(* PLC project CM, Beckhoff Automation GmbH TwinCAT PLC Control 3.5.13.21 *)
(* stored: creationDateTime 2024-07-22T16:12:49.8021823, modificationDateTime 2024-07-22T16:12:49.8062692 *)

TYPE E_AnalysisIDs :
(
	(* analysis chain *)
	eID_Source := 1,
	
	// Magnetude Spectrum
	eID_MagSpectrum,	
	eID_MagSpec_Sink, 
	
	// RMS intergrate
	eID_RMS,	
	eID_RMS_Sink,
	
	// Envelope Spectrum
	eID_EnvSpectrum,	
	eID_EnvSpec_Sink,
	
	// Envelope 
	eID_Env,	
	eID_Env_Sink	
	
) UDINT;
END_TYPE

TYPE ST_HRErrHist :
STRUCT
{attribute 'displaymode':='hex'}
	hrErrCode	: HRESULT;
	sErrSource	: STRING(63);
	nErrCount	: UDINT;
END_STRUCT
END_TYPE

FUNCTION_BLOCK FB_HRErrHist
(* v1.10
build up an error history consisting of two arrays and one index.
The index shows the actual array position. The last error id and the count for this id are saved in the arrays.
If an error id is the same as the previous input error the counter is increased. Otherwise the index is increased.
*)
VAR_INPUT
	bEdgeDetect	: BOOL;	(* FALSE: every input(bErr) is processed; TRUE: only rising edge of input is processed *)
END_VAR
VAR_OUTPUT
	nErrSum		: UINT;
	nErrIdx		: UINT; // error list index of last occured error (max. cHistLen)
	aErrList	: ARRAY[1..cHistLen] OF ST_HRErrHist;
END_VAR

VAR
	bNewErr		: BOOL;
	fbErrTrig	: R_TRIG;
END_VAR
VAR CONSTANT
	cHistLen	: UINT := 100;
END_VAR

                  
                

METHOD AddError
VAR_INPUT
	bErr		: BOOL;
	hrErrCode	: HRESULT;
	sErrSource	: STRING(63);
END_VAR
                        fbErrTrig(CLK:=bErr);
IF bEdgeDetect THEN
	bNewErr := fbErrTrig.Q;
ELSE
	bNewErr := bErr;
END_IF

IF bNewErr THEN
	nErrSum := nErrSum + 1;
	IF nErrIdx < cHistLen THEN
		IF nErrIdx = 0 THEN
			nErrIdx	:= nErrIdx + 1;
		ELSIF aErrList[nErrIdx].hrErrCode <> hrErrCode OR aErrList[nErrIdx].sErrSource <> sErrSource THEN
			nErrIdx	:= nErrIdx + 1;
		END_IF
		aErrList[nErrIdx].hrErrCode := hrErrCode;
		aErrList[nErrIdx].sErrSource := sErrSource;
		aErrList[nErrIdx].nErrCount := aErrList[nErrIdx].nErrCount + 1;
	END_IF
END_IF

                      
END_METHOD

METHOD Reset
VAR_INPUT
END_VAR
                        nErrSum := 0;
nErrIdx := 0;
MEMSET(ADR(aErrList),0,SIZEOF(aErrList));
                      
END_METHOD
END_FUNCTION_BLOCK

FUNCTION_BLOCK FB_SystemTime
VAR_INPUT
END_VAR
VAR_OUTPUT
END_VAR
VAR
	GetLocalSystemTime 	: FB_LocalSystemTime;
	wDateW				: WORD;
END_VAR

                  GetLocalSystemTime(bEnable := TRUE);
                

PROPERTY dtDateTimeFull : DT
GET
VAR
END_VAR
                          dtDateTimeFull 	:= SYSTEMTIME_TO_DT(GetLocalSystemTime.systemTime);
                        
END_GET
END_PROPERTY

PROPERTY sDate : STRING
GET
VAR
END_VAR
                          sDate	:= MID(sDateTimeFull,10,1);
                        
END_GET
END_PROPERTY

PROPERTY sDateTime : STRING
GET
VAR
END_VAR
                          sDateTime := MID(sDateTimeFull,19,1);
                        
END_GET
END_PROPERTY

PROPERTY sDateTimeFull : STRING
GET
VAR
END_VAR
                          sDateTimeFull 	:= SYSTEMTIME_TO_STRING(GetLocalSystemTime.systemTime);
                        
END_GET
END_PROPERTY

PROPERTY sDayOfWeek : STRING
GET
VAR
END_VAR
                          wDateW	:=  GetLocalSystemTime.systemTime.wDayOfWeek;
IF wDateW = 0 THEN
	sDayOfWeek := 'Sunday';
ELSIF wDateW = 1 THEN
	sDayOfWeek := 'Monday';
ELSIF wDateW = 2 THEN
	sDayOfWeek := 'Tuesday';
ELSIF wDateW = 3 THEN
	sDayOfWeek := 'Wednesday';
ELSIF wDateW = 4 THEN
	sDayOfWeek := 'Thursday';
ELSIF wDateW = 5 THEN
	sDayOfWeek := 'Friday';
ELSIF wDateW = 6 THEN
	sDayOfWeek := 'Saturday';
END_IF
                        
END_GET
END_PROPERTY

PROPERTY sTime : STRING
GET
VAR
END_VAR
                          sTime := MID(sDateTimeFull,8,12);
                        
END_GET
END_PROPERTY

PROPERTY wDay : Word
GET
VAR
END_VAR
                          wDay :=  GetLocalSystemTime.systemTime.wDay;
                        
END_GET
END_PROPERTY

PROPERTY wHour : WORD
GET
VAR
END_VAR
                          wHour	:=	GetLocalSystemTime.systemTime.wHour;
                        
END_GET
END_PROPERTY

PROPERTY wMilliSeconds : WORD
GET
VAR
END_VAR
                          wMilliseconds	:=	GetLocalSystemTime.systemTime.wMilliseconds;
                        
END_GET
END_PROPERTY

PROPERTY wMinute : WORD
GET
VAR
END_VAR
                          wMinute	:=	GetLocalSystemTime.systemTime.wMinute;
                        
END_GET
END_PROPERTY

PROPERTY wMonth : Word
GET
VAR
END_VAR
                          wMonth	:=  GetLocalSystemTime.systemTime.wMonth;
                        
END_GET
END_PROPERTY

PROPERTY wSecond : WORD
GET
VAR
END_VAR
                          wSecond	:=	GetLocalSystemTime.systemTime.wSecond;
                        
END_GET
END_PROPERTY

PROPERTY wYear : Word
GET
VAR
END_VAR
                          wYear :=  GetLocalSystemTime.systemTime.wYear;
                        
END_GET
END_PROPERTY
END_FUNCTION_BLOCK

PROGRAM MAIN
VAR
	nSample				: UDINT;
	
	fbSource			: FB_CMA_Source := (	stInitPars 	:= cInitSource, 
												nOwnID 		:= eID_Source, 
												aDestIDs 	:= [eID_MagSpectrum,
																eID_EnvSpectrum,
																eID_Env,
																eID_RMS]);		
										
	fbSinkMagSpec		: FB_CMA_Sink 	:= ( 	nOwnID 		:= eID_MagSpec_Sink);
	fbSinkEnvSpec		: FB_CMA_Sink 	:= ( 	nOwnID 		:= eID_EnvSpec_Sink);
	fbSinkEnv			: FB_CMA_Sink 	:= ( 	nOwnID 		:= eID_Env_Sink);
	fbSinkRMS			: FB_CMA_Sink 	:= ( 	nOwnID 		:= eID_RMS_Sink); 
	
	nChannelIdx			: UDINT;

	k, m, l: UDINT;
	nChnIdx: UDINT;
END_VAR

                  Source();
Sink();
// input from EL3632
FOR nChannelIdx := 1 TO cMaxChannels DO
	FOR k := 1 TO cOversamples DO
		aAccBuffer[nChannelIdx][k] 		:= INT_TO_LREAL(aEl3632[nChannelIdx][k])*(5/EXPT(2,15))/(0.1)*9.81;
	END_FOR	
END_FOR


                

ACTION Sink:
                      // Push results to sink

fbSinkMagSpec.Output2DStd(	pDataOut 	:= ADR(aMagSpecResult), 
					nDataOutSize 		:= SIZEOF(aMagSpecResult), 
					eElementType 		:= eMA_TypeCode_LREAL, 
					nOptionPars			:= 0);
				
fbSinkEnvSpec.Output2DStd(	pDataOut 	:= ADR(aEnvSpecResult), 
					nDataOutSize 		:= SIZEOF(aEnvSpecResult), 
					eElementType 		:= eMA_TypeCode_LREAL, 
					nOptionPars			:= 0); 
					
fbSinkEnv.Output2DStd(	pDataOut 		:= ADR(aEnvResult), 
					nDataOutSize 		:= SIZEOF(aEnvResult), 
					eElementType 		:= eMA_TypeCode_LREAL, 
					nOptionPars			:= 0); 								
				
fbSinkRMS.Output2DStd(	pDataOut 		:= ADR(aRMSResult), 
					nDataOutSize 		:= SIZEOF(aRMSResult), 
					eElementType 		:= eMA_TypeCode_LREAL, 
					nOptionPars			:= 0); 						
			
                    
END_ACTION

ACTION Source:
                      fbSource.Input2DStd( pDataIn 			:= ADR(aAccBuffer),
				  nDataInSize 			:= SIZEOF(aAccBuffer), 
				  eElementType 			:= eMA_TypeCode_LREAL,
				  nOptionPars			:= cCMA_Option_MarkInterruption ); 

                    
END_ACTION
END_PROGRAM

PROGRAM MAIN_CM
VAR
	fbMagSpec			: FB_CMA_MagnitudeSpectrum 
						:= (	stInitPars 	:= cInitSpectrum, 
								nOwnID 		:= eID_MagSpectrum, 
								aDestIDs 	:= [eID_MagSpec_Sink] ); 
										
	fbEnvSpec			: FB_CMA_EnvelopeSpectrum 
						:= ( 	stInitPars 	:= cInitEnvSpec, 
								nOwnID 		:= eID_EnvSpectrum, 
								aDestIDs 	:= [eID_EnvSpec_Sink] );	
								
	fbEnv				: FB_CMA_Envelope 
						:= ( 	stInitPars 	:= cInitEnv, 
								nOwnID 		:= eID_Env, 
								aDestIDs 	:= [eID_Env_Sink] );	
								
	fbRMS				: FB_CMA_IntegratedRMS
						:= ( 	stInitPars	:= cInitIRMS,
								nOwnID		:= eID_RMS,
								aDestIDs	:= [eID_RMS_Sink]);
		
	nErrorID			: UDINT;
	fbErrHist			: FB_HRErrHist; 
	hrErrList			: ARRAY[1..2] OF HRESULT;
	bPause				: BOOL;
	
END_VAR

                  IF NOT bPause THEN
//
END_IF

PRG_Database();
PRG_Motor_Sensor();

fbMagSpec.Call();
fbEnvSpec.Call();
fbEnv.Call();

fbRMS.Call();
//fbHistArray.CallEx(nAppendData := cAppendData, bResetData := bResetHist);

                
END_PROGRAM

PROGRAM PRG_Calculate
VAR
	nChnIdx, i, k		: UDINT;
	m, n, p, j, l, q	: UDINT:= 1;
	fSumRMSEnv			: LREAL;
END_VAR

                  FOR nChnIdx := 1 TO cMaxChannels DO
	// Calculate Frequency
	fSampleRate								:= cOversamples * (1000.0 / fSampleTaskCycleTime);
	fResolution 							:= fSampleRate / cFFTLength;	
	
	// Calculate velocity spectrum                              	     	
	FOR i := 1 TO cFFTResult DO             	
		fFrequency[nChnIdx][i]				:= (i - 1) * fResolution;			
		IF i <> 1 THEN
			aVeloSpecResult[nChnIdx][i]		:= aMagSpecResult[nChnIdx][i]/(2*PI*fFrequency[nChnIdx][i])*1000;
		ELSE
			aVeloSpecResult[nChnIdx][i]		:= 0;
		END_IF
	END_FOR
	
	//Calculate RMS of Envelope
	fSumRMSEnv 								:= 0;
	FOR p := 1 TO cBufferLength DO
		fSumRMSEnv							:= fSumRMSEnv + EXPT(aEnvResult[nChnIdx][p],2);
	END_FOR
	aRmsEnvResult[nChnIdx]					:= SQRT(fSumRMSEnv/cBufferLength);
	
	//Scale up for HMI 
	IF m < cScaleHMI THEN
		FOR n := 1 TO cOversamples DO
			aTWFBuffer[nChnIdx][(m-1)*10+n]		:= aAccBuffer[nChnIdx][n];   
		END_FOR
		m										:= m + 1;
	ELSE
		m										:= cScaleHMI;
		FOR l := 1 TO cScaleHMI-1 DO
			FOR n := 1 TO cOversamples DO
				aTWFBuffer[nChnIdx][(l-1)*10+n]	:= aTWFBuffer[nChnIdx][(l)*10+n];   
			END_FOR
		END_FOR
		FOR q := 1 TO cOversamples DO
			aTWFBuffer[nChnIdx][(m-1)*10+q]		:= aAccBuffer[nChnIdx][q];   
		END_FOR	
	END_IF	
	
END_FOR

IF aTime[cOversamples*cScaleHMI] <> cOversamples*cScaleHMI THEN
	FOR k := 1 TO cOversamples*cScaleHMI DO aTime[k] := k; END_FOR
END_IF






                
END_PROGRAM

PROGRAM PRG_Database
VAR
	fbSystemTime			:	FB_SystemTime;
	bSaveData				: BOOL;
	bLoadData				: BOOL;
	nStateSave, nStateLoad	: INT;
	tTimer1, tTimer2		: TON;
	bTest					: BOOL;
	nStateADS				: INT;
END_VAR

                  fbSystemTime();
sCurrentTime	:= fbSystemTime.sTime;
nCurrentSec		:= fbSystemTime.wSecond;
CASE nStateSave OF
	0:
		tTimer1(IN := FALSE);
		IF nCurrentSec = 70 OR sCurrentTime = '06:00:00' OR sCurrentTime = '14:00:00' OR sCurrentTime = '22:00:00' THEN
			nStateSave			:= 1;
		END_IF
	1:
		aFFTAcceleration1Add		:= aMagSpecResult[1];
		aFFTVelocity1Add			:= aVeloSpecResult[1];
		aFFTEnvelope1Add			:= aEnvSpecResult[1];
		RMSAcc1Add					:= aRMSResult[1][1]/9.81;
		RMSVel1Add					:= aRMSResult[1][2]*1000;
		RMSEnv1Add					:= aRMSEnvResult[1]/9.81;
		
		aFFTAcceleration2Add		:= aMagSpecResult[2];
		aFFTVelocity2Add			:= aVeloSpecResult[2];
		aFFTEnvelope2Add			:= aEnvSpecResult[2];
		RMSAcc2Add					:= aRMSResult[2][1]/9.81;
		RMSVel2Add					:= aRMSResult[2][2]*1000;
		RMSEnv2Add					:= aRMSEnvResult[2]/9.81;		
		bAddData					:= TRUE;
		nStateSave					:= 2;
	2:
		IF NOT bAddData THEN
			tTimer1(IN := TRUE,PT := T#2S);
			IF tTimer1.Q THEN
				nStateSave			:= 0;		
			END_IF	
		END_IF
			
		
END_CASE

CASE nStateADS OF
	0:
		IF bCheckADS THEN
			nStateADS := 1;
		ELSE
			tTimer2(IN := TRUE,PT := T#5S);
			IF tTimer2.Q THEN
				nStateADS := 2;
			END_IF
		END_IF
		
	1:
		bCheckADS := FALSE;
		bError	:= FALSE;
		tTimer2(IN := FALSE);
		nStateADS := 0;
	2:
		bError := TRUE;
		tTimer2(IN := FALSE);
		IF bCheckADS THEN
			nStateADS := 0;
		END_IF
END_CASE
                
END_PROGRAM

PROGRAM PRG_Motor_Sensor
VAR
END_VAR

                  IF bMotorRun THEN
//	wMotorRun	:= 18;
ELSE
//	wMotorRun	:= 1;
END_IF

IF fFreq >= 0 AND fFreq <= 60 THEN
	wFreq		:= REAL_TO_WORD(fFreq*100);
END_IF
                
END_PROGRAM

CONFIGURATION Application
  RESOURCE CM ON PLC
(* global variable list CM_Params *)
VAR_GLOBAL CONSTANT
	cOversamples 		: UDINT 	:= 10;		// number of oversamples
	cMaxChannels		: UDINT		:= 2;
	cOrder				: UDINT		:= 1;		// Maximum order of integration: 0 = acceleration, 1 = velocity, 2 = place. 
	cBufferLength		: UDINT		:= 1600;	// buffer size
	cWindowLength		: UDINT		:= 3200;	// internal buffer size with 50% overlapping
	cRMSBuffer     		: UDINT 	:= 4800;  	// e.g. keep 2 old buffers in mind and add one new buffer to calc RMS value	
	cFFTResult 			: UDINT 	:= 2049;	// result of mag. spectrum (cFFTLength/2+1)
	cFFTLength			: UDINT		:= 4096;	// length of FFT for mag. spectrum	
	cScaleHMI			: UDINT     := 50;
	cWindowParameters	: T_CM_WindowParameters := [0.0, 0.0, 0.0, 0.0, 0.0];	
	
    cInitSource			: ST_MA_MultiArray_InitPars 
						:= ( 	eTypeCode 			:= eMA_TypeCode_LREAL, 
								nDims 				:= 2, 
								aDimSizes 			:= [cMaxChannels,cBufferLength]);	
	
	cInitSpectrum 		: ST_CM_MagnitudeSpectrum_InitPars 
						:= (	nFFT_Length 		:= cFFTLength, 
								nWindowLength 		:= cWindowLength,
								nChannels			:= cMaxChannels,
								bTransformToDecibel	:= FALSE, 
								eWindowType 		:= E_CM_WindowType.eCM_HannWindow, 
								nOverlap			:= cWindowLength/2,
								eScalingType 		:= E_CM_ScalingType.eCM_RMS);
								
	cInitEnvSpec 		: ST_CM_EnvelopeSpectrum_InitPars 
						:= (	nFFT_Length			:= cFFTLength,
								nWindowLength		:= cWindowLength,
								nChannels			:= cMaxChannels,
								bTransformToDecibel	:= FALSE,
								fDecibelThreshold	:= cCM_MinArgLog10, 
								eWindowType			:= eCM_HannWindow,  
								nOverlap			:= cWindowLength/2,         
								eScalingType 		:= eCM_RMS);   
								
	cInitEnv	 		: ST_CM_Envelope_InitPars 
						:= (	nFFT_Length			:= cFFTLength,
								nWindowLength		:= cWindowLength,
								nChannels			:= cMaxChannels);   	
		
	cInitIRMS			: ST_CM_IntegratedRMS_InitPars
						:= ( 	nFFT_Length			:= cFFTLength,
								nWindowLength		:= cWindowLength,
								fSampleRate			:= 10000,
								fLowerFrequencyLimit	:= 20.0,
								fUpperFrequencyLimit	:= 4000.0,
								nMaxBands			:= 1,
								nOrder				:= cOrder,
								nChannels			:= cMaxChannels,
								eWindowType			:= E_CM_WindowType.eCM_HannWindow,
								nOverlap			:=  cWindowLength/2,
								bTransformToDecibel	:= FALSE);
					
END_VAR

VAR_GLOBAL
	fSampleTaskCycleTime		: LREAL := 1; 	// ms
	fSampleRate					: LREAL; 		// Hz  ( sample rate = oversampling factor / cycle time )
	fResolution					: LREAL; 		// Hz/Idx	
	aAccAlarm					: ARRAY[1..cMaxChannels] OF LREAL;
	aVeloAlarm					: ARRAY[1..cMaxChannels] OF LREAL;
	aEnvAlarm					: ARRAY[1..cMaxChannels] OF LREAL;
	
	aAccWarning					: ARRAY[1..cMaxChannels] OF LREAL;
	aVeloWarning				: ARRAY[1..cMaxChannels] OF LREAL;
	aEnvWarning					: ARRAY[1..cMaxChannels] OF LREAL;
	
	nCurrentDate				: WORD;
	sCurrentTime				: STRING;
	nCurrentHour				: WORD;
	nCurrentSec					: WORD;
	
END_VAR
(* global variable list CM_Data *)
VAR_GLOBAL

	aAccBuffer			: ARRAY[1..cMaxChannels] OF ARRAY[1..cOversamples] OF LREAL;   	
		
	aMagSpecResult		: ARRAY[1..cMaxChannels] OF ARRAY[1..cFFTResult] OF LREAL;	
	aVeloSpecResult		: ARRAY[1..cMaxChannels] OF ARRAY[1..cFFTResult] OF LREAL;
	aEnvSpecResult		: ARRAY[1..cMaxChannels] OF ARRAY[1..cFFTResult] OF LREAL;
	
	aEnvResult			: ARRAY[1..cMaxChannels] OF ARRAY[1..cBufferLength] OF LREAL;
		
	aRMSResult			: ARRAY[1..cMaxChannels] OF ARRAY[1..cOrder+1] OF LREAL;
	aRMSEnvResult		: ARRAY[1..cMaxChannels] OF LREAL;

	fFrequency			: ARRAY[1..cMaxChannels] OF ARRAY[1..cFFTResult] OF LREAL; 		// Hz	
	aTWFBuffer			: ARRAY[1..cMaxChannels] OF ARRAY[1..cOversamples*cScaleHMI] OF LREAL;  
	aTime				: ARRAY[1..cOversamples*cScaleHMI] OF UDINT;	
END_VAR
(* global variable list GVL_ADS *)
VAR_GLOBAL
	aFFTAcceleration1Add 	: ARRAY[1..cFFTResult] OF LREAL;
	aFFTVelocity1Add 		: ARRAY[1..cFFTResult] OF LREAL;
	aFFTEnvelope1Add 		: ARRAY[1..cFFTResult] OF LREAL;
	RMSAcc1Add				: LREAL;
	RMSVel1Add				: LREAL;
	RMSEnv1Add				: LREAL;
	Temperature1Add			: REAL;
	//point_2
	aFFTAcceleration2Add 	: ARRAY[1..cFFTResult] OF LREAL;
	aFFTVelocity2Add 		: ARRAY[1..cFFTResult] OF LREAL;
	aFFTEnvelope2Add 		: ARRAY[1..cFFTResult] OF LREAL;
	RMSAcc2Add				: LREAL;
	RMSVel2Add				: LREAL;
	RMSEnv2Add				: LREAL;
	Temperature2Add			: REAL;
	//bAdd
	bAddData				: BOOL;
	bCheckADS				: BOOL;
	bError					: BOOL;
END_VAR
(* global variable list GVL_IO *)
VAR_GLOBAL
	aEl3632 AT %I*		: ARRAY[1..cMaxChannels] OF ARRAY[1..cOversamples] OF INT;	// Input from hardware e.g. EL3632	
	wMotorRun	AT %Q*	: WORD;
	wFreq		AT %Q*	: WORD;
	bRev		AT %I*	: BOOL;
	bMotorRun			: BOOL;
	fFreq				: REAL;
END_VAR
    TASK PlcTask(INTERVAL := T#0ms, PRIORITY := 4);
    TASK PlcTaskCM(INTERVAL := T#0ms, PRIORITY := 10);
    TASK TaskCalc(INTERVAL := T#0ms, PRIORITY := 8);
    PROGRAM MAIN WITH PlcTask : MAIN;
    PROGRAM MAIN_CM WITH PlcTaskCM : MAIN_CM;
    PROGRAM PRG_Calculate WITH TaskCalc : PRG_Calculate;
  END_RESOURCE
END_CONFIGURATION
